TYPE rotaryKnifeSpeedCurve_TypeConfig :
STRUCT
	
	machineSpeed	: REAL := 150;
	sheetLength		: REAL	:= 800;

END_STRUCT
END_TYPE

(* stored: Version 1.1.0.1
   DUT rotaryKnifeSpeedCurve_TypeConfig: Id {b3b36856-d758-4ea4-8c9c-e858c00923c4} *)
